FUNCTION_BLOCK EventQueue EXTENDS Queue
VAR_INPUT
END_VAR
VAR_OUTPUT
	{attribute 'OPC.UA.DA' := '1'}
    {attribute 'OPC.UA.DA.StructuredType' := '1'}
	ErrorEvent:EventReport_Typ;		
END_VAR
VAR
	{attribute 'OPC.UA.DA' := '0'}
	EventActiveFlag:BOOL;
	{attribute 'OPC.UA.DA' := '0'}
	InitDone:		BOOL;
	{attribute 'OPC.UA.DA' := '0'}
    SubsystemIDString:	STRING;

END_VAR
VAR_STAT
	{attribute 'OPC.UA.DA' := '0'}
	SequentialID:	DINT;
END_VAR

IF NOT InitDone THEN
	mInit();
	InitDone:= TRUE;
END_IF
IF THIS^.EntriesCount > 0 AND (THIS^.CheckQReadAvailable()) AND EventActiveFlag=FALSE  THEN
	EventActiveFlag:=TRUE;
    THIS^.Dequeue(ADR(ErrorEvent),SIZEOF(ErrorEvent));
	SequentialID := SequentialID + 1 ;
	IF SequentialID >= 16#7FFFFFFF THEN
		SequentialID := 0;
	END_IF

	ErrorEvent.SequentialID := SequentialID;
	SubsystemIDString := TO_STRING(ErrorEvent.SubsysID);
	LogError_v2('Send event %s from %s, FlowID %d, SequentialID %d ' ,
		ErrorEvent.EventID, SubsystemIDString, ErrorEvent.FlowID,SequentialID,dint_0,dint_0,dint_0,dint_0,dint_0,dint_0);
END_IF

{attribute 'TcRpcEnable':='1'}
METHOD mAckEvent : BOOL
VAR_INPUT
END_VAR
EventActiveFlag:=FALSE;
MEMSET(ADR(ErrorEvent),0,SIZEOF(ErrorEvent));

mAckEvent := TRUE;
END_METHOD

{attribute 'TcRpcEnable':='1'}
METHOD mClearQueue : BOOL
VAR_INPUT
END_VAR
 THIS^.Clear();
 LogError_v2('Clear EventQueue ' ,dint_0, dint_0, dint_0,dint_0,dint_0,dint_0,dint_0,dint_0,dint_0,dint_0);
END_METHOD

METHOD mInit : BOOL
VAR_INPUT
END_VAR
SetLoggerCategoryName('Events');
END_METHOD

END_FUNCTION_BLOCK

(* stored: Version 1.1.0.1, ProductVersion 3.1.4024.3
   POU EventQueue: Id {e457a2c8-e0cd-0fde-002a-0340784a6446}, SpecialFunc None
   Method mAckEvent: Id {325148e9-2bf4-0fae-0a25-9f6e39847a39}
   Method mClearQueue: Id {510c58b2-5aa5-4b63-9f92-12d1775c553d}
   Method mInit: Id {88550928-d113-46f8-a064-a847369073bb} *)
